// TIA Portal V20 export
TYPE "LKinCtrl_PointEditor_typePointTableInternalEvents"
// stored: Access Published
   STRUCT
      updateTable { ExternalAccessible := 'False'; ExternalVisible := 'False'; ExternalWritable := 'False'} : Bool;   // triggers internal event. Reset internally.
   END_STRUCT;
END_TYPE
